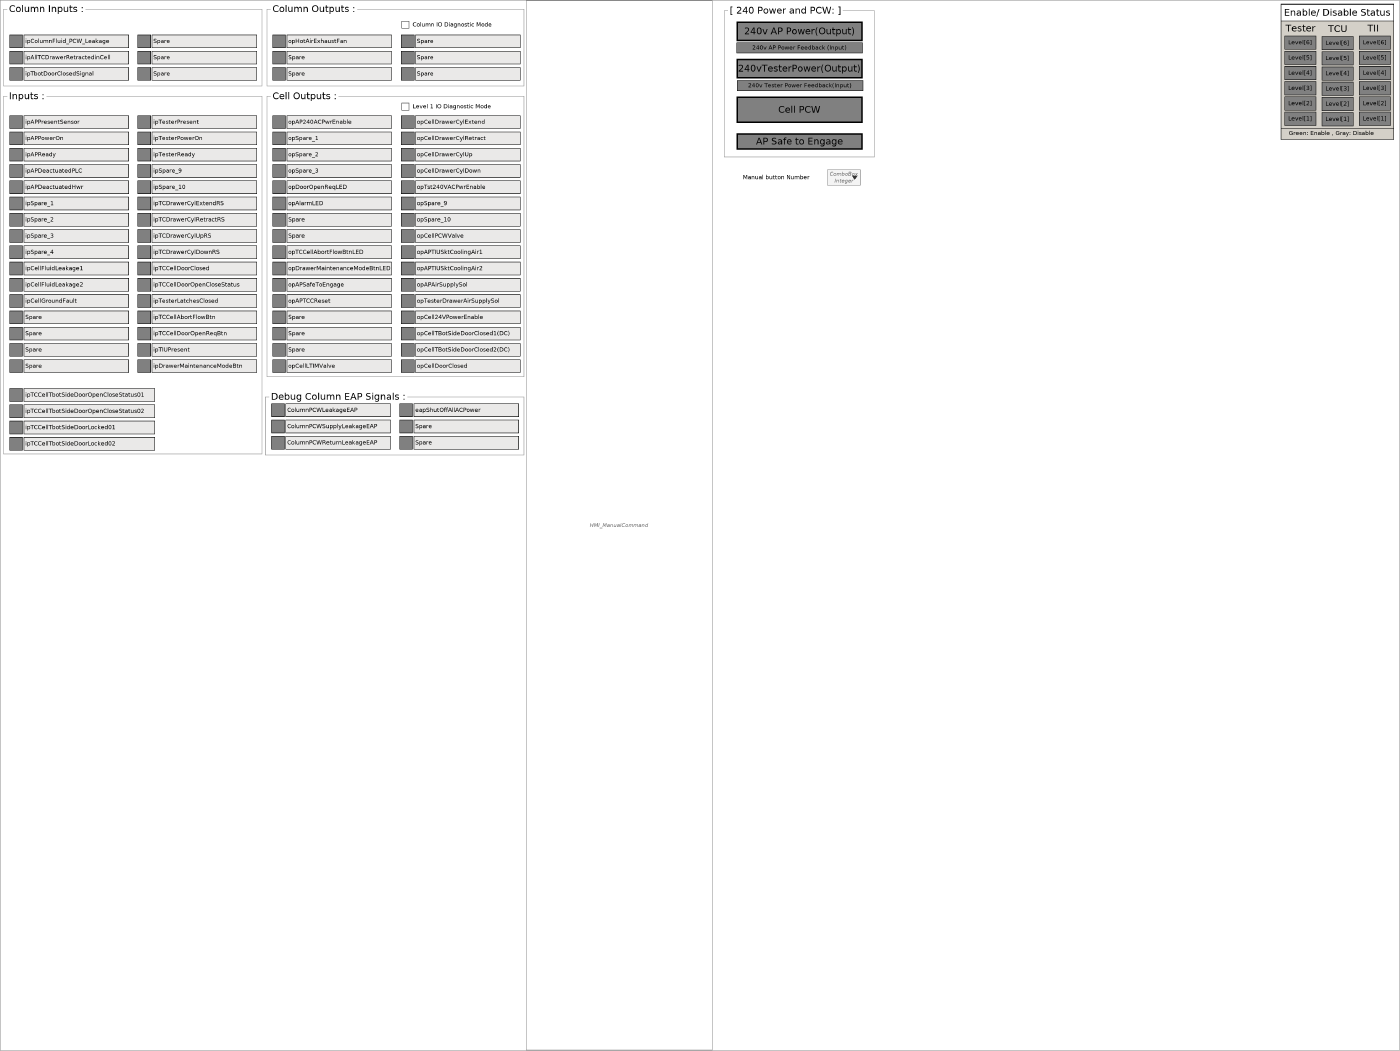
VISUALIZATION HMI_All_Level  // 2667x2003
    GroupBox (1379,12 287x287), "[ 240 Power and PCW: ]"
        RoundedRectangle (24,69 240x20), "240v AP Power Feedback (Input)", colour toggle: arrTCMultiLevel[iHMICbLevelSelection].fbTCMultiLevelSeq.stMLDIO.ipAPPowerOn
        RoundedRectangle (25,141 240x20), "240v Tester Power Feedback(Input)", colour toggle: arrTCMultiLevel[iHMICbLevelSelection].fbTCMultiLevelSeq.stMLDIO.ipTesterPowerOn
        RoundedRectangle (24,242 240x31), "AP Safe to Engage", colour toggle: arrTCMultiLevel[iHMICbLevelSelection].fbTCMultiLevelSeq.stMLDIO.opAPSafeToEngage
    GroupBox (6,175 493x690), "Inputs :"
        RoundedRectangle (12,510 25x25)
        RoundedRectangle (256,510 25x25), colour toggle: arrTCMultiLevel[iHMICbLevelSelection].fbTCMultiLevelSeq.stMLDIO.ipDrawerMaintenanceModeBtn
    GroupBox (508,175 490x543), "Cell Outputs :"
        RoundedRectangle (283,45 200x25), "opCellDrawerCylExtend"
            toggle arrTCMultiLevel[iHMICbLevelSelection].fbTCMultiLevelSeq.stMLDIO.opCellDrawerCylExtend
        RoundedRectangle (38,479 200x25), "Spare"
    RoundedRectangle (546,220 200x25), "opAP240ACPwrEnable"
        toggle arrTCMultiLevel[iHMICbLevelSelection].fbTCMultiLevelSeq.stMLDIO.opAP240ACPwrEnable
    RoundedRectangle (546,251 200x25), "opSpare_1"
        toggle arrTCMultiLevel[iHMICbLevelSelection].fbTCMultiLevelSeq.stMLDIO.opSpare_1
    RoundedRectangle (546,282 200x25), "opSpare_2"
        toggle arrTCMultiLevel[iHMICbLevelSelection].fbTCMultiLevelSeq.stMLDIO.opSpare_2
    RoundedRectangle (546,313 200x25), "opSpare_3"
        toggle arrTCMultiLevel[iHMICbLevelSelection].fbTCMultiLevelSeq.stMLDIO.opSpare_3
    RoundedRectangle (546,344 200x25), "opDoorOpenReqLED"
        toggle arrTCMultiLevel[iHMICbLevelSelection].fbTCMultiLevelSeq.stMLDIO.opDoorOpenReqLED
    RoundedRectangle (546,375 200x25), "opAlarmLED"
        toggle arrTCMultiLevel[iHMICbLevelSelection].fbTCMultiLevelSeq.stMLDIO.opAlarmLED
    RoundedRectangle (546,406 200x25), "Spare"
    RoundedRectangle (546,437 200x25), "Spare"
    RoundedRectangle (546,468 200x25), "opTCCellAbortFlowBtnLED"
        toggle arrTCMultiLevel[iHMICbLevelSelection].fbTCMultiLevelSeq.stMLDIO.opTCCellAbortFlowBtnLED
    RoundedRectangle (546,499 200x25), "opDrawerMaintenanceModeBtnLED"
        toggle arrTCMultiLevel[iHMICbLevelSelection].fbTCMultiLevelSeq.stMLDIO.opDrawerMaintenanceModeBtnLED
    RoundedRectangle (546,530 200x25), "opAPSafeToEngage"
        toggle arrTCMultiLevel[iHMICbLevelSelection].fbTCMultiLevelSeq.stMLDIO.opAPSafeToEngage
    RoundedRectangle (546,561 200x25), "opAPTCCReset"
        toggle arrTCMultiLevel[iHMICbLevelSelection].fbTCMultiLevelSeq.stMLDIO.opAPTCCReset
    RoundedRectangle (546,592 200x25), "Spare"
    RoundedRectangle (546,623 200x25), "Spare"
    RoundedRectangle (791,654 200x25), "opCellTBotSideDoorClosed2(DC)"
        toggle arrTCMultiLevel[iHMICbLevelSelection].fbTCMultiLevelSeq.stMLDIO.opCellTBOtSideDoorClosed2
    RoundedRectangle (546,685 200x25), "opCellLTIMValve"
        toggle arrTCMultiLevel[iHMICbLevelSelection].fbTCMultiLevelSeq.stMLDIO.opCellLTIMValve
    RoundedRectangle (519,220 25x25), colour toggle: arrTCMultiLevel[iHMICbLevelSelection].fbTCMultiLevelSeq.stMLDIO.opAP240ACPwrEnable
    RoundedRectangle (519,251 25x25), colour toggle: arrTCMultiLevel[iHMICbLevelSelection].fbTCMultiLevelSeq.stMLDIO.opSpare_1
    RoundedRectangle (519,282 25x25), colour toggle: arrTCMultiLevel[iHMICbLevelSelection].fbTCMultiLevelSeq.stMLDIO.opSpare_2
    RoundedRectangle (519,313 25x25), colour toggle: arrTCMultiLevel[iHMICbLevelSelection].fbTCMultiLevelSeq.stMLDIO.opSpare_3
    RoundedRectangle (519,344 25x25), colour toggle: arrTCMultiLevel[iHMICbLevelSelection].fbTCMultiLevelSeq.stMLDIO.opDoorOpenReqLED
    RoundedRectangle (519,375 25x25), colour toggle: arrTCMultiLevel[iHMICbLevelSelection].fbTCMultiLevelSeq.stMLDIO.opAlarmLED
    RoundedRectangle (519,406 25x25)
    RoundedRectangle (519,437 25x25)
    RoundedRectangle (519,468 25x25), colour toggle: arrTCMultiLevel[iHMICbLevelSelection].fbTCMultiLevelSeq.stMLDIO.opTCCellAbortFlowBtnLED
    RoundedRectangle (519,499 25x25), colour toggle: arrTCMultiLevel[iHMICbLevelSelection].fbTCMultiLevelSeq.stMLDIO.opDrawerMaintenanceModeBtnLED
    RoundedRectangle (519,530 25x25), colour toggle: arrTCMultiLevel[iHMICbLevelSelection].fbTCMultiLevelSeq.stMLDIO.opAPSafeToEngage
    RoundedRectangle (519,561 25x25), colour toggle: arrTCMultiLevel[iHMICbLevelSelection].fbTCMultiLevelSeq.stMLDIO.opAPTCCReset
    RoundedRectangle (519,592 25x25)
    RoundedRectangle (519,623 25x25)
    RoundedRectangle (519,654 25x25)
    RoundedRectangle (519,685 25x25), colour toggle: arrTCMultiLevel[iHMICbLevelSelection].fbTCMultiLevelSeq.stMLDIO.opCellLTIMValve
    RoundedRectangle (45,220 200x25), "ipAPPresentSensor"
    RoundedRectangle (45,251 200x25), "ipAPPowerOn"
    RoundedRectangle (45,282 200x25), "ipAPReady"
    RoundedRectangle (45,313 200x25), "ipAPDeactuatedPLC"
    RoundedRectangle (45,344 200x25), "ipAPDeactuatedHwr"
    RoundedRectangle (45,375 200x25), "ipSpare_1"
    RoundedRectangle (45,406 200x25), "ipSpare_2"
    RoundedRectangle (45,437 200x25), "ipSpare_3"
    RoundedRectangle (45,468 200x25), "ipSpare_4"
    RoundedRectangle (45,499 200x25), "ipCellFluidLeakage1"
    RoundedRectangle (45,530 200x25), "ipCellFluidLeakage2"
    RoundedRectangle (45,561 200x25), "ipCellGroundFault"
    RoundedRectangle (45,592 200x25), "Spare"
    RoundedRectangle (45,623 200x25), "Spare"
    RoundedRectangle (45,654 200x25), "Spare"
    RoundedRectangle (45,685 200x25), "Spare"
    RoundedRectangle (18,220 25x25), colour toggle: arrTCMultiLevel[iHMICbLevelSelection].fbTCMultiLevelSeq.stMLDIO.ipAPPresentSensor
    RoundedRectangle (18,251 25x25), colour toggle: arrTCMultiLevel[iHMICbLevelSelection].fbTCMultiLevelSeq.stMLDIO.ipAPPowerOn
    RoundedRectangle (18,282 25x25), colour toggle: arrTCMultiLevel[iHMICbLevelSelection].fbTCMultiLevelSeq.stMLDIO.ipAPReady
    RoundedRectangle (18,313 25x25), colour toggle: arrTCMultiLevel[iHMICbLevelSelection].fbTCMultiLevelSeq.stMLDIO.ipHandlerSafeToEnterPLC
    RoundedRectangle (18,344 25x25), colour toggle: arrTCMultiLevel[iHMICbLevelSelection].fbTCMultiLevelSeq.stMLDIO.ipHandlerSafeToEnterHwr
    RoundedRectangle (18,375 25x25), colour toggle: arrTCMultiLevel[iHMICbLevelSelection].fbTCMultiLevelSeq.stMLDIO.ipSpare_1
    RoundedRectangle (18,406 25x25), colour toggle: arrTCMultiLevel[iHMICbLevelSelection].fbTCMultiLevelSeq.stMLDIO.ipSpare_2
    RoundedRectangle (18,437 25x25), colour toggle: arrTCMultiLevel[iHMICbLevelSelection].fbTCMultiLevelSeq.stMLDIO.ipSpare_3
    RoundedRectangle (18,468 25x25), colour toggle: arrTCMultiLevel[iHMICbLevelSelection].fbTCMultiLevelSeq.stMLDIO.ipSpare_4
    RoundedRectangle (18,499 25x25), colour toggle: arrTCMultiLevel[iHMICbLevelSelection].fbTCMultiLevelSeq.stMLDIO.ipCellFluidLeakage1
    RoundedRectangle (18,530 25x25), colour toggle: arrTCMultiLevel[iHMICbLevelSelection].fbTCMultiLevelSeq.stMLDIO.ipCellFluidLeakage2
    RoundedRectangle (18,561 25x25), colour toggle: arrTCMultiLevel[iHMICbLevelSelection].fbTCMultiLevelSeq.stMLDIO.ipCellGroundFault
    RoundedRectangle (18,592 25x25)
    RoundedRectangle (18,623 25x25)
    RoundedRectangle (18,654 25x25)
    RoundedRectangle (791,251 200x25), "opCellDrawerCylRetract"
        toggle arrTCMultiLevel[iHMICbLevelSelection].fbTCMultiLevelSeq.stMLDIO.opCellDrawerCylRetract
    RoundedRectangle (791,282 200x25), "opCellDrawerCylUp"
        toggle arrTCMultiLevel[iHMICbLevelSelection].fbTCMultiLevelSeq.stMLDIO.opCellDrawerCylUp
    RoundedRectangle (791,313 200x25), "opCellDrawerCylDown"
        toggle arrTCMultiLevel[iHMICbLevelSelection].fbTCMultiLevelSeq.stMLDIO.opCellDrawerCylDown
    RoundedRectangle (791,344 200x25), "opTst240VACPwrEnable"
        toggle arrTCMultiLevel[iHMICbLevelSelection].fbTCMultiLevelSeq.stMLDIO.opTst240VACPwrEnable
    RoundedRectangle (791,375 200x25), "opSpare_9"
        toggle arrTCMultiLevel[iHMICbLevelSelection].fbTCMultiLevelSeq.stMLDIO.opSpare_9
    RoundedRectangle (791,406 200x25), "opSpare_10"
        toggle arrTCMultiLevel[iHMICbLevelSelection].fbTCMultiLevelSeq.stMLDIO.opSpare_10
    RoundedRectangle (791,437 200x25), "opCellPCWValve"
        toggle arrTCMultiLevel[iHMICbLevelSelection].fbTCMultiLevelSeq.stMLDIO.opCellPCWValve
    RoundedRectangle (791,468 200x25), "opAPTIUSktCoolingAir1"
        toggle arrTCMultiLevel[iHMICbLevelSelection].fbTCMultiLevelSeq.stMLDIO.opTIUSktAirSol_1
    RoundedRectangle (791,499 200x25), "opAPTIUSktCoolingAir2"
        toggle arrTCMultiLevel[iHMICbLevelSelection].fbTCMultiLevelSeq.stMLDIO.opTIUSktAirSol_2
    RoundedRectangle (791,530 200x25), "opAPAirSupplySol"
        toggle arrTCMultiLevel[iHMICbLevelSelection].fbTCMultiLevelSeq.stMLDIO.opAPAirSupplySol
    RoundedRectangle (791,561 200x25), "opTesterDrawerAirSupplySol"
        toggle arrTCMultiLevel[iHMICbLevelSelection].fbTCMultiLevelSeq.stMLDIO.opTesterDrawerAirSupplySol
    RoundedRectangle (791,592 200x25), "opCell24VPowerEnable"
        toggle arrTCMultiLevel[iHMICbLevelSelection].fbTCMultiLevelSeq.stMLDIO.opCell24VPowerEnable
    RoundedRectangle (791,623 200x25), "opCellTBotSideDoorClosed1(DC)"
        toggle arrTCMultiLevel[iHMICbLevelSelection].fbTCMultiLevelSeq.stMLDIO.opCellTBOtSideDoorClosed1
    RoundedRectangle (791,685 200x25), "opCellDoorClosed"
        toggle arrTCMultiLevel[iHMICbLevelSelection].fbTCMultiLevelSeq.stMLDIO.opCellDoorClosed
    RoundedRectangle (764,220 25x25), colour toggle: arrTCMultiLevel[iHMICbLevelSelection].fbTCMultiLevelSeq.stMLDIO.opCellDrawerCylExtend
    RoundedRectangle (764,251 25x25), colour toggle: arrTCMultiLevel[iHMICbLevelSelection].fbTCMultiLevelSeq.stMLDIO.opCellDrawerCylRetract
    RoundedRectangle (764,282 25x25), colour toggle: arrTCMultiLevel[iHMICbLevelSelection].fbTCMultiLevelSeq.stMLDIO.opCellDrawerCylUp
    RoundedRectangle (764,313 25x25), colour toggle: arrTCMultiLevel[iHMICbLevelSelection].fbTCMultiLevelSeq.stMLDIO.opCellDrawerCylDown
    RoundedRectangle (764,344 25x25), colour toggle: arrTCMultiLevel[iHMICbLevelSelection].fbTCMultiLevelSeq.stMLDIO.opTst240VACPwrEnable
    RoundedRectangle (764,375 25x25), colour toggle: arrTCMultiLevel[iHMICbLevelSelection].fbTCMultiLevelSeq.stMLDIO.opSpare_9
    RoundedRectangle (764,406 25x25), colour toggle: arrTCMultiLevel[iHMICbLevelSelection].fbTCMultiLevelSeq.stMLDIO.opSpare_10
    RoundedRectangle (764,437 25x25), colour toggle: arrTCMultiLevel[iHMICbLevelSelection].fbTCMultiLevelSeq.stMLDIO.opCellPCWValve
    RoundedRectangle (764,468 25x25), colour toggle: arrTCMultiLevel[iHMICbLevelSelection].fbTCMultiLevelSeq.stMLDIO.opTIUSktAirSol_1
    RoundedRectangle (764,499 25x25), colour toggle: arrTCMultiLevel[iHMICbLevelSelection].fbTCMultiLevelSeq.stMLDIO.opTIUSktAirSol_2
    RoundedRectangle (764,530 25x25), colour toggle: arrTCMultiLevel[iHMICbLevelSelection].fbTCMultiLevelSeq.stMLDIO.opAPAirSupplySol
    RoundedRectangle (764,561 25x25), colour toggle: arrTCMultiLevel[iHMICbLevelSelection].fbTCMultiLevelSeq.stMLDIO.opTesterDrawerAirSupplySol
    RoundedRectangle (764,592 25x25), colour toggle: arrTCMultiLevel[iHMICbLevelSelection].fbTCMultiLevelSeq.stMLDIO.opCell24VPowerEnable
    RoundedRectangle (764,623 25x25), colour toggle: arrTCMultiLevel[iHMICbLevelSelection].fbTCMultiLevelSeq.stMLDIO.opCellTBOtSideDoorClosed1
    RoundedRectangle (764,654 25x25), colour toggle: arrTCMultiLevel[iHMICbLevelSelection].fbTCMultiLevelSeq.stMLDIO.opCellTBOtSideDoorClosed2
    RoundedRectangle (764,685 25x25), colour toggle: arrTCMultiLevel[iHMICbLevelSelection].fbTCMultiLevelSeq.stMLDIO.opCellDoorClosed
    RoundedRectangle (289,220 200x25), "ipTesterPresent"
    RoundedRectangle (289,251 200x25), "ipTesterPowerOn"
    RoundedRectangle (289,282 200x25), "ipTesterReady"
    RoundedRectangle (289,313 200x25), "ipSpare_9"
    RoundedRectangle (289,344 200x25), "ipSpare_10"
    RoundedRectangle (289,375 200x25), "ipTCDrawerCylExtendRS"
    RoundedRectangle (289,406 200x25), "ipTCDrawerCylRetractRS"
    RoundedRectangle (289,437 200x25), "ipTCDrawerCylUpRS"
    RoundedRectangle (289,468 200x25), "ipTCDrawerCylDownRS"
    RoundedRectangle (289,499 200x25), "ipTCCellDoorClosed"
    RoundedRectangle (289,530 200x25), "ipTCCellDoorOpenCloseStatus"
    RoundedRectangle (289,561 200x25), "ipTesterLatchesClosed"
    RoundedRectangle (289,592 200x25), "ipTCCellAbortFlowBtn"
    RoundedRectangle (289,623 200x25), "ipTCCellDoorOpenReqBtn"
    RoundedRectangle (289,654 200x25), "ipTIUPresent"
    RoundedRectangle (289,685 200x25), "ipDrawerMaintenanceModeBtn"
    RoundedRectangle (262,220 25x25), colour toggle: arrTCMultiLevel[iHMICbLevelSelection].fbTCMultiLevelSeq.stMLDIO.ipTesterPresent
    RoundedRectangle (262,251 25x25), colour toggle: arrTCMultiLevel[iHMICbLevelSelection].fbTCMultiLevelSeq.stMLDIO.ipTesterPowerOn
    RoundedRectangle (262,282 25x25), colour toggle: arrTCMultiLevel[iHMICbLevelSelection].fbTCMultiLevelSeq.stMLDIO.ipTesterReady
    RoundedRectangle (262,313 25x25), colour toggle: arrTCMultiLevel[iHMICbLevelSelection].fbTCMultiLevelSeq.stMLDIO.ipSpare_9
    RoundedRectangle (262,344 25x25), colour toggle: arrTCMultiLevel[iHMICbLevelSelection].fbTCMultiLevelSeq.stMLDIO.ipSpare_10
    RoundedRectangle (262,375 25x25), colour toggle: arrTCMultiLevel[iHMICbLevelSelection].fbTCMultiLevelSeq.stMLDIO.ipTCDrawerCylExtendRS
    RoundedRectangle (262,406 25x25), colour toggle: arrTCMultiLevel[iHMICbLevelSelection].fbTCMultiLevelSeq.stMLDIO.ipTCDrawerCylRetractRS
    RoundedRectangle (262,437 25x25), colour toggle: arrTCMultiLevel[iHMICbLevelSelection].fbTCMultiLevelSeq.stMLDIO.ipTCDrawerCylUpRS
    RoundedRectangle (262,468 25x25), colour toggle: arrTCMultiLevel[iHMICbLevelSelection].fbTCMultiLevelSeq.stMLDIO.ipTCDrawerCylDownRS
    RoundedRectangle (262,499 25x25), colour toggle: arrTCMultiLevel[iHMICbLevelSelection].fbTCMultiLevelSeq.stMLDIO.ipTCCellDoorClosed
    RoundedRectangle (262,530 25x25), colour toggle: arrTCMultiLevel[iHMICbLevelSelection].fbTCMultiLevelSeq.stMLDIO.ipTCCellDoorOpenCloseStatus
    RoundedRectangle (262,561 25x25), colour toggle: arrTCMultiLevel[iHMICbLevelSelection].fbTCMultiLevelSeq.stMLDIO.ipTesterLatchesClosed
    RoundedRectangle (262,592 25x25), colour toggle: arrTCMultiLevel[iHMICbLevelSelection].fbTCMultiLevelSeq.stMLDIO.ipTCCellAbortFlowBtn
    RoundedRectangle (262,623 25x25), colour toggle: arrTCMultiLevel[iHMICbLevelSelection].fbTCMultiLevelSeq.stMLDIO.ipTCCellDoorOpenReqBtn
    RoundedRectangle (262,654 25x25), colour toggle: arrTCMultiLevel[iHMICbLevelSelection].fbTCMultiLevelSeq.stMLDIO.ipTIUPresent
    Checkbox (763,188 200x30), "Level 1 IO Diagnostic Mode", variable: arrTCMultiLevel[iHMICbLevelSelection].fbTCMultiLevelSeq.stMLVIO.bDiagnosticMode, input disabled if: TRUE
    GroupBox (6,9 493x155), "Column Inputs :"
    GroupBox (508,9 490x155), "Column Outputs :"
        RoundedRectangle (283,57 200x25), "Spare"
    RoundedRectangle (546,66 200x25), "opHotAirExhaustFan"
        toggle fbTCColumn.stTCColumnDIO.opHotAirExhaustFan
    RoundedRectangle (546,97 200x25), "Spare"
    RoundedRectangle (546,128 200x25), "Spare"
    RoundedRectangle (519,66 25x25), colour toggle: fbTCColumn.stTCColumnDIO.opHotAirExhaustFan
    RoundedRectangle (519,97 25x25)
    RoundedRectangle (519,128 25x25)
    RoundedRectangle (45,66 200x25), "ipColumnFluid_PCW_Leakage"
    RoundedRectangle (45,97 200x25), "ipAllTCDrawerRetractedinCell"
    RoundedRectangle (45,128 200x25), "ipTbotDoorClosedSignal"
    RoundedRectangle (18,66 25x25), colour toggle: fbTCColumn.stTCColumnDIO.ipColumnFluid_PCW_Leakage
    RoundedRectangle (18,97 25x25), colour toggle: fbTCColumn.stTCColumnDIO.ipAllTCDrawerRetractedinCell
    RoundedRectangle (18,128 25x25), colour toggle: fbTCColumn.stTCColumnDIO.ipTbotDoorClosedSignal
    RoundedRectangle (791,97 200x25), "Spare"
    RoundedRectangle (791,128 200x25), "Spare"
    RoundedRectangle (764,66 25x25)
    RoundedRectangle (764,97 25x25)
    RoundedRectangle (764,128 25x25)
    RoundedRectangle (289,66 200x25), "Spare"
    RoundedRectangle (289,97 200x25), "Spare"
    RoundedRectangle (289,128 200x25), "Spare"
    RoundedRectangle (262,66 25x25)
    RoundedRectangle (262,97 25x25)
    RoundedRectangle (262,128 25x25)
    Checkbox (763,32 200x30), "Column IO Diagnostic Mode", variable: bColIODiagnosticsMode
    RoundedRectangle (45,740 250x25), "ipTCCellTbotSideDoorOpenCloseStatus01"
    RoundedRectangle (45,771 250x25), "ipTCCellTbotSideDoorOpenCloseStatus02"
    RoundedRectangle (45,802 250x25), "ipTCCellTbotSideDoorLocked01"
    RoundedRectangle (45,833 250x25), "ipTCCellTbotSideDoorLocked02"
    RoundedRectangle (18,740 25x25), colour toggle: arrTCMultiLevel[iHMICbLevelSelection].fbTCMultiLevelSeq.stMLDIO.ipTCCellTbotSideDoorOpenCloseStatus01
    RoundedRectangle (18,771 25x25), colour toggle: arrTCMultiLevel[iHMICbLevelSelection].fbTCMultiLevelSeq.stMLDIO.ipTCCellTbotSideDoorOpenCloseStatus02
    RoundedRectangle (18,802 25x25), colour toggle: arrTCMultiLevel[iHMICbLevelSelection].fbTCMultiLevelSeq.stMLDIO.ipTCCellTbotSideDoorLocked01
    RoundedRectangle (18,833 25x25), colour toggle: arrTCMultiLevel[iHMICbLevelSelection].fbTCMultiLevelSeq.stMLDIO.ipTCCellTbotSideDoorLocked02
    GroupBox (505,748 493x119), "Debug Column EAP Signals :"
    RoundedRectangle (544,769 200x25), "ColumnPCWLeakageEAP"
    RoundedRectangle (544,800 200x25), "ColumnPCWSupplyLeakageEAP"
    RoundedRectangle (544,831 200x25), "ColumnPCWReturnLeakageEAP"
    RoundedRectangle (517,769 25x25), colour toggle: fbTCColumn.stTCColumnDIO.eapDColumnPCWLeakage
    RoundedRectangle (517,800 25x25), colour toggle: fbTCColumn.stTCColumnDIO.eapDColumnPCWSupplyLeakage
    RoundedRectangle (517,831 25x25), colour toggle: fbTCColumn.stTCColumnDIO.eapDColumnPCWReturnLeakage
    RoundedRectangle (788,769 200x25), "eapShutOffAllACPower", colour toggle: eapShutOffAllACPower
    RoundedRectangle (788,800 200x25), "Spare"
    RoundedRectangle (788,831 200x25), "Spare"
    RoundedRectangle (761,769 25x25), colour toggle: eapShutOffAllACPower
    RoundedRectangle (761,800 25x25)
    RoundedRectangle (761,831 25x25)
    Frame (1002,1 355x2000), invisible if: Not bEnableManualCommandTest1 AND Not bEnableManualCommandTest2
        shows HMI_ManualCommand()
    RoundedRectangle (1403,41 240x37), "240v AP Power(Output)", colour toggle: arrTCMultiLevel[iHMICbLevelSelection].fbTCMultiLevelSeq.stMLDIO.opAP240ACPwrEnable
    RoundedRectangle (1403,112 240x37), "240vTesterPower(Output)", colour toggle: arrTCMultiLevel[iHMICbLevelSelection].fbTCMultiLevelSeq.stMLDIO.opTst240VACPwrEnable
    RoundedRectangle (1403,184 240x50), "Cell PCW", colour toggle: arrTCMultiLevel[iHMICbLevelSelection].fbTCMultiLevelSeq.stMLDIO.opCellPCWValve
    Group (2440,7 225x262)
        Rectangle (0,0 215x259)
        Rectangle (0,237 215x22)
        RoundedRectangle (7,206 60x26), "Level[1]", tooltip "VIO Status", colour toggle: TC_ModuleState[1].Tester = E_State.eEnabled
        RoundedRectangle (7,177 60x26), "Level[2]", tooltip "VIO Status", colour toggle: TC_ModuleState[2].Tester= E_State.eEnabled
        RoundedRectangle (7,148 60x26), "Level[3]", tooltip "VIO Status", colour toggle: TC_ModuleState[3].Tester = E_State.eEnabled
        RoundedRectangle (7,119 60x26), "Level[4]", tooltip "VIO Status", colour toggle: TC_ModuleState[4].Tester = E_State.eEnabled
        RoundedRectangle (7,90 60x26), "Level[5]", tooltip "VIO Status", colour toggle: TC_ModuleState[5].Tester = E_State.eEnabled
        RoundedRectangle (7,61 60x26), "Level[6]", tooltip "VIO Status", colour toggle: TC_ModuleState[6].Tester = E_State.eEnabled
        Label (6,32 61x30), "Tester"
        RoundedRectangle (149,206 60x26), "Level[1]", tooltip "VIO Status", colour toggle: TC_ModuleState[1].TCSite[1].TIERII = E_State.eEnabled
        RoundedRectangle (149,177 60x26), "Level[2]", tooltip "VIO Status", colour toggle: TC_ModuleState[2].TCSite[1].TIERII = E_State.eEnabled
        RoundedRectangle (149,148 60x26), "Level[3]", tooltip "VIO Status", colour toggle: TC_ModuleState[3].TCSite[1].TIERII = E_State.eEnabled
        RoundedRectangle (149,119 60x26), "Level[4]", tooltip "VIO Status", colour toggle: TC_ModuleState[4].TCSite[1].TIERII = E_State.eEnabled
        RoundedRectangle (149,90 60x26), "Level[5]", tooltip "VIO Status", colour toggle: TC_ModuleState[5].TCSite[1].TIERII = E_State.eEnabled
        RoundedRectangle (149,61 60x26), "Level[6]", tooltip "VIO Status", colour toggle: TC_ModuleState[6].TCSite[1].TIERII = E_State.eEnabled
        Label (162,32 32x30), "TII"
        RoundedRectangle (78,207 60x26), "Level[1]", tooltip "VIO Status", colour toggle: TC_ModuleState[1].TCSite[1].TCU = E_State.eEnabled
        RoundedRectangle (78,178 60x26), "Level[2]", tooltip "VIO Status", colour toggle: TC_ModuleState[2].TCSite[1].TCU= E_State.eEnabled
        RoundedRectangle (78,149 60x26), "Level[3]", tooltip "VIO Status", colour toggle: TC_ModuleState[3].TCSite[1].TCU = E_State.eEnabled
        RoundedRectangle (78,120 60x26), "Level[4]", tooltip "VIO Status", colour toggle: TC_ModuleState[4].TCSite[1].TCU = E_State.eEnabled
        RoundedRectangle (78,91 60x26), "Level[5]", tooltip "VIO Status", colour toggle: TC_ModuleState[5].TCSite[1].TCU = E_State.eEnabled
        RoundedRectangle (78,62 60x26), "Level[6]", tooltip "VIO Status", colour toggle: TC_ModuleState[6].TCSite[1].TCU = E_State.eEnabled
        Label (87,33 43x30), "TCU"
        Label (12,232 213x30), "Green: Enable , Gray: Disable"
        Rectangle (0,1 215x32), "Enable/ Disable Status"
    ComboBoxInteger (1576,323 63x30), variable: TestManually.iBtnNo
    Label (1404,323 149x30), "Manual button Number"
END_VISUALIZATION

(* stored: Version 1.1.0.1, ProductVersion 3.1.4022.18
   Visu HMI_All_Level: Id {f5088c06-5310-4ef7-bef4-63100f837b86} *)
